(* CODESYS project InfiniteStateMachine
   Author: Roy Ratcliffe
   Company: Roy Ratcliffe
   DefaultNamespace: ISM
   DocFormat: reStructuredText
   LanguageModelAttribute: qualified-access-only
   Placeholder: ISML
   Title: Infinite State Machine Library
   Version: 0.1.1.1

Project tree, tasks and I/O mapping:
  InfiniteStateMachine/
    Enums/
    Function Blocks/
      function block StateMachine [ST]: AtLevel, Depth, Enter, GoTo, In, Jump, Leave, Pop, Push, Top
    Functions/
      function DepthOfState [ST]
      function IsSameState [ST]
      function Topology [ST]
    GlobalConstants/
      global variables ISM
    Interfaces/
      interface IState: Enter, Leave, SuperState
    Structs/
    Types/
      data type IStateArray
  Library Information/
    function GetLibVersion [ST]
    function GetLibVersionNumber [ST]
    function IsLibReleased [ST]
*)

// InfiniteStateMachine/Types/IStateArray
TYPE
	IStateArray : ARRAY[0..ISM.gc_iMaxDepth] OF IState;
END_TYPE

// InfiniteStateMachine/GlobalConstants/ISM
{attribute 'qualified_only'}
VAR_GLOBAL CONSTANT
	gc_iMaxDepth : INT := 7;
END_VAR

// Library Information/GetLibVersion
// This function has been automatically generated from the project information.
FUNCTION GetLibVersion : VERSION
VAR_INPUT
	
END_VAR

GetLibVersion.uiMajor := 0;
GetLibVersion.uiMinor := 1;
GetLibVersion.uiServicePack := 1;
GetLibVersion.uiPatch := 1;

END_FUNCTION

// Library Information/GetLibVersionNumber
// This function has been automatically generated from the project information.
FUNCTION GetLibVersionNumber : DWORD
VAR_INPUT
	
END_VAR

GetLibVersionNumber := 65793;

END_FUNCTION

// Library Information/IsLibReleased
// This function has been automatically generated from the project information.
FUNCTION IsLibReleased : BOOL
VAR_INPUT
	
END_VAR

IsLibReleased := FALSE;

END_FUNCTION

// InfiniteStateMachine/Function Blocks/StateMachine
FUNCTION_BLOCK FINAL StateMachine
VAR_INPUT
END_VAR
VAR_OUTPUT
END_VAR
VAR
	itfStates : IStateArray;
	iDepth : INT := 0;
END_VAR

METHOD PUBLIC AtLevel : IState
VAR_INPUT
	iLevel : INT;
END_VAR
IF 0 <= iLevel AND iLevel < iDepth THEN
	AtLevel := itfStates[iLevel];
END_IF
END_METHOD

METHOD Depth : INT
VAR_INPUT
END_VAR
Depth := iDepth;
END_METHOD

METHOD PROTECTED Enter
VAR_INPUT
	itfState : IState;
END_VAR
IF Push(itfState) THEN
	itfState.Enter(THIS^);
END_IF
END_METHOD

METHOD PUBLIC GoTo
VAR_INPUT
	itfState : IState;
END_VAR
VAR
	fbStateMachine : StateMachine;
	iDepth : INT := 0;
END_VAR
fbStateMachine.Jump(itfState);
WHILE iDepth < Depth() AND iDepth < fbStateMachine.Depth() AND IsSameState(AtLevel(iDepth), fbStateMachine.AtLevel(iDepth)) DO
	iDepth := iDepth + 1;
END_WHILE
WHILE Depth() > iDepth DO
	Leave();
END_WHILE
WHILE fbStateMachine.Depth() > iDepth DO
	Enter(fbStateMachine.AtLevel(iDepth));
	iDepth := iDepth + 1;
END_WHILE
END_METHOD

METHOD In : BOOL
VAR_INPUT
	itfState: IState;
END_VAR
VAR
	iLevel : INT := 0;
END_VAR
(*
 * The following do-while loop's condition assumes early-out semantics.
 * It assumes that the second sub-condition does *not* evaluate unless the first sub-condition is true.
 *)
WHILE iLevel < iDepth AND itfStates[iLevel] <> itfState DO
	iLevel := iLevel + 1;
END_WHILE
In := iLevel < iDepth;
END_METHOD

METHOD Jump
VAR_INPUT
	itfState : IState;
END_VAR
iDepth := DepthOfState(itfState, ISM.gc_iMaxDepth, itfStates);
END_METHOD

METHOD PROTECTED Leave
VAR_INPUT
END_VAR
VAR
	itfState : IState;
END_VAR
itfState := Pop();
IF itfState <> 0 THEN
	itfState.Leave(THIS^);
END_IF
END_METHOD

METHOD PROTECTED Pop : IState
VAR_INPUT
END_VAR
IF iDepth > 0 THEN
	iDepth := iDepth - 1;
	Pop := itfStates[iDepth];
    (*
     * Clear the popped state from the stack. This is not strictly necessary,
     * but it can help catch use-after-free bugs.
     *)
	itfStates[iDepth] := 0;
ELSE
	Pop := 0;
END_IF
END_METHOD

METHOD PROTECTED Push : BOOL
VAR_INPUT
	itfState : IState;
END_VAR
Push := iDepth < ISM.gc_iMaxDepth;
IF Push THEN
	itfStates[iDepth] := itfState;
	iDepth := iDepth + 1;
END_IF
END_METHOD

METHOD PUBLIC Top : IState
VAR_INPUT
END_VAR
IF iDepth > 0 THEN
	Top := itfStates[iDepth - 1];
END_IF
END_METHOD

END_FUNCTION_BLOCK

// InfiniteStateMachine/Interfaces/IState
INTERFACE IState EXTENDS __SYSTEM.IQueryInterface

METHOD Enter
VAR_INPUT
	fbStateMachine : StateMachine;
END_VAR
END_METHOD

METHOD Leave
VAR_INPUT
	fbStateMachine : StateMachine;
END_VAR
END_METHOD

PROPERTY SuperState : IState
GET
END_GET
SET
END_SET
END_PROPERTY

END_INTERFACE

// InfiniteStateMachine/Functions/IsSameState
FUNCTION IsSameState : BOOL
VAR_INPUT
	itfStateLHS : IState;
	itfStateRHS : IState;
END_VAR
VAR
END_VAR

IsSameState := itfStateLHS = itfStateRHS;

END_FUNCTION

// InfiniteStateMachine/Functions/DepthOfState
{attribute 'suppress_warning' := '0561'}
FUNCTION DepthOfState : INT
VAR_INPUT
	itfState : IState;
	iDepth : INT;
	itfStates : REFERENCE TO IStateArray;
END_VAR
VAR
END_VAR

IF itfState = 0 THEN
	DepthOfState := 0;
ELSE
	DepthOfState := Topology(itfState, iDepth, itfStates);
END_IF

END_FUNCTION

// InfiniteStateMachine/Functions/Topology
{attribute 'suppress_warning' := '0561'}
FUNCTION Topology : INT
VAR_INPUT
	itfState : IState;
	iDepth : INT;
	itfStates : REFERENCE TO IStateArray;
END_VAR
VAR
END_VAR

IF iDepth = 0 THEN
	Topology := 0;
ELSE
	Topology := DepthOfState(itfState.SuperState, iDepth - 1, itfStates);
	itfStates[Topology] := itfState;
	Topology := Topology + 1;
END_IF

END_FUNCTION
